TYPE typeOutputArea :
STRUCT
    OutPorToWhiSigAreAll : UINT;
    NumericalDataFlag    : UINT;
    StartFlag            : USINT;
    OperationMethod      : USINT;
    Speed                : UINT;
    TargetPosition       : DINT;
    Acceleration         : UINT;
    Deceleration         : UINT;
    PushingForce         : UINT;
    TriggerLv            : UINT;
    PushingSpeed         : UINT;
    PushingForceForPos   : UINT;
    Area1                : DINT;
    Area2                : DINT;
    PositioningWidth     : DINT;
END_STRUCT
END_TYPE

(* stored: Version 1.1.0.1, ProductVersion 3.1.4024.6
   DUT typeOutputArea: Id {0cb5db62-1e6e-48c7-b7b6-b27880dffc6a} *)
